(* PLC project 이름이 없는, 알려지지 않은 이름이 없는 1 *)
(* stored: creationDateTime 2024-07-08T18:26:42, modificationDateTime 2024-07-08T19:55:30 *)

PROGRAM program0
  VAR
    PBS AT %IX0.0 : BOOL;
    EMS AT %IX0.1 : BOOL;
    PS1 AT %IX0.2 : BOOL;
    PS2 AT %IX0.3 : BOOL;
    PS3 AT %IX0.4 : BOOL;
    IS1 AT %IX0.5 : BOOL;
    CONV AT %QX0.0 : BOOL;
    CYN AT %QX0.1 : BOOL;
    RL AT %QX0.2 : BOOL;
    YL AT %QX0.3 : BOOL;
    GL AT %QX0.4 : BOOL;
    SEQUENCE_1 AT %MX0.0 : BOOL;
    SEQUENCE_2 AT %MX0.1 : BOOL;
    SEQUENCE_3 AT %MX0.2 : BOOL;
    RST AT %MX0.4 : BOOL;
    SEQUENCE_4 AT %MX0.3 : BOOL;
    IS_METAL AT %MX0.5 : BOOL;
    IS_NON_METAL AT %MX0.6 : BOOL;
    FLICKER AT %MX1.0 : BOOL;
    SEQ_WAIT AT %MX1.1 : BOOL;
    SEQ_WAIT_2 AT %MX1.2 : BOOL;
  END_VAR
  VAR
    TON0 : TON;
    TON1 : TON;
    TON2 : TON;
    TON3 : TON;
    TON4 : TON;
    TON5 : TON;
  END_VAR

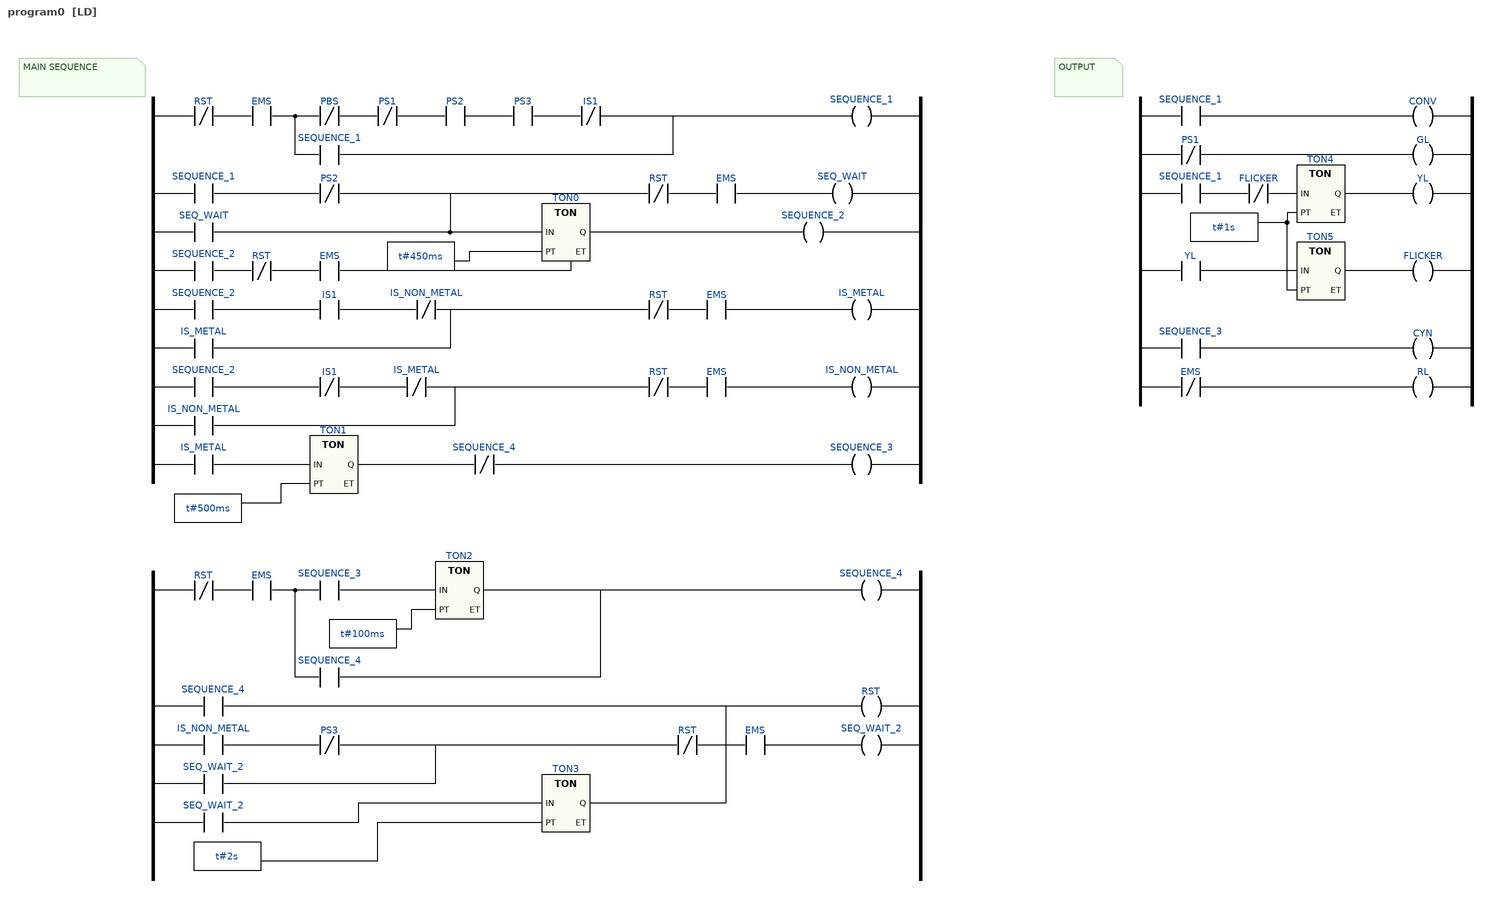
(* LD diagram, written out as Structured Text *)
(* MAIN SEQUENCE *)
(* OUTPUT *)
SEQUENCE_1 := NOT RST AND EMS AND (SEQUENCE_1 OR NOT PBS AND NOT PS1 AND PS2 AND PS3 AND NOT IS1);
CONV := SEQUENCE_1;
TON0(IN := SEQ_WAIT, PT := t#450ms);
SEQUENCE_2 := TON0.Q OR SEQUENCE_2 AND NOT RST AND EMS;
IS_METAL := (SEQUENCE_2 AND IS1 AND NOT IS_NON_METAL OR IS_METAL) AND NOT RST AND EMS;
TON1(IN := IS_METAL, PT := t#500ms);
SEQUENCE_3 := TON1.Q AND NOT SEQUENCE_4;
TON2(IN := NOT RST AND EMS AND SEQUENCE_3, PT := t#100ms);
SEQUENCE_4 := TON2.Q OR NOT RST AND EMS AND SEQUENCE_4;
TON3(IN := SEQ_WAIT_2, PT := t#2s);
RST := SEQUENCE_4 OR TON3.Q;
IS_NON_METAL := (SEQUENCE_2 AND NOT IS1 AND NOT IS_METAL OR IS_NON_METAL) AND NOT RST AND EMS;
GL := NOT PS1;
RL := NOT EMS;
TON4(IN := SEQUENCE_1 AND NOT FLICKER, PT := t#1s);
YL := TON4.Q;
TON5(IN := YL, PT := t#1s);
FLICKER := TON5.Q;
SEQ_WAIT := (SEQ_WAIT OR SEQUENCE_1 AND NOT PS2) AND NOT RST AND EMS;
SEQ_WAIT_2 := (SEQ_WAIT_2 OR IS_NON_METAL AND NOT PS3) AND NOT RST AND EMS;
CYN := SEQUENCE_3;
END_PROGRAM

CONFIGURATION Config0
  RESOURCE Res0 ON PLC
    TASK task0(INTERVAL := T#20ms, PRIORITY := 0);
    PROGRAM instance0 WITH task0 : program0;
  END_RESOURCE
END_CONFIGURATION
